FUNCTION_BLOCK SpindleCIA402Velocity IMPLEMENTS SpindleController
VAR
	// CIA402 Control word
	oControlWord AT %Q*: ST_CIA402ControlWord;
	// CIA402 Status word
	iStatusWord AT %I*: UINT;
	// CIA402 actual velocity parameter
	iActualVelocity AT %I* : UDINT;
	// CIA402 target velocity
	oTargetVelocity AT %Q* : INT;
	// Forward/backward is specified by positive or negative speed
	VelocityMultiplier : INT := 1;
END_VAR

(* Return the current speed of the spindle in RPM*)
METHOD GetSpeed : UDINT
GetSpeed := iActualVelocity;
END_METHOD

METHOD GetState : E_CIA402State
VAR CONSTANT
	NotReadyToSwitchOnValue : UINT := 2#0000_0000_0000_0000;
	NotReadyToSwitchOnMask : UINT := 2#0000_0000_0100_1111;
	SwitchOnDisabledValue : UINT := 2#0000_0000_0100_0000;
	SwitchOnDisabledMask : UINT := NotReadyToSwitchOnMask;
	ReadyToSwitchOnValue : UINT := 2#0000_0000_0010_0001;
	ReadyToSwitchOnMask : UINT := 2#0000_0000_0110_1111;
	SwitchedOnValue : UINT := 2#0000_0000_0010_0011;
	SwitchedOnMask : UINT := ReadyToSwitchOnMask;
	OperationEnabledValue : UINT := 2#0000_0000_0010_0111;
	OperationEnabledMask : UINT := ReadyToSwitchOnMask;
	QuickStopActiveValue : UINT := 2#0000_0000_0000_0111;
	QuickStopActiveMask : UINT := ReadyToSwitchOnMask;
	FaultReactionActiveValue : UINT := 2#0000_0000_0000_1111;
	FaultReactionActiveMask : UINT := 2#0000_0000_0100_1111;
	FaultValue : UINT := 2#0000_0000_0000_1000;
	FaultMask : UINT := FaultReactionActiveMask;
END_VAR
IF (iStatusWord AND NotReadyToSwitchOnMask) = NotReadyToSwitchOnValue THEN
	GetState := E_CIA402State.NotReadyToSwitchOn;
ELSIF (iStatusWord AND SwitchOnDisabledMask) = SwitchOnDisabledValue THEN
	GetState := E_CIA402State.SwitchOnDisabled;
ELSIF (iStatusWord AND ReadyToSwitchOnMask) = ReadyToSwitchOnValue THEN
	GetState := E_CIA402State.ReadyToSwitchOn;
ELSIF (iStatusWord AND SwitchedOnMask) = SwitchedOnValue THEN
	GetState := E_CIA402State.SwitchedOn;
ELSIF (iStatusWord AND OperationEnabledMask) = OperationEnabledValue THEN
	GetState := E_CIA402State.OperationEnabled;
ELSIF (iStatusWord AND QuickStopActiveMask) = QuickStopActiveValue THEN
	GetState := E_CIA402State.QuickStopActive;
ELSIF (iStatusWord AND FaultReactionActiveMask) = FaultReactionActiveValue THEN
	GetState := E_CIA402State.FaultReactionActive;
ELSIF (iStatusWord AND FaultMask) = FaultValue THEN
	GetState := E_CIA402State.Fault;
ELSE
	GetState := E_CIA402State.Unknown_State;
END_IF
END_METHOD

METHOD GetStatus : ST_CIA402StatusWord
VAR_INPUT
END_VAR
MEMCPY(ADR(GetStatus), ADR(iStatusWord), SIZEOF(iStatusWord));
END_METHOD

METHOD HasFault : BOOL
VAR_INPUT
END_VAR
HasFault := GetState() = E_CIA402State.Fault OR GetState() = E_CIA402State.FaultReactionActive;
END_METHOD

METHOD Run : BOOL
oControlWord.FaultReset := FALSE;
CASE GetState() OF
	E_CIA402State.SwitchOnDisabled:
		oControlWord.EnableVoltage := TRUE;
	E_CIA402State.ReadyToSwitchOn:
		oControlWord.SwitchOn := TRUE;
	E_CIA402State.SwitchedOn:
		oControlWord.EnableOperation := TRUE;
	// We don't need explicit fault handling. 
	// The fault will cause the controller to tell the drive to stop, 
	// and the stop will take care of the fault reset.
END_CASE
END_METHOD

METHOD SetDirection : BOOL
VAR_INPUT
	(* Set the spindle rotation direction*)
	Reverse	: BOOL;
END_VAR
IF Reverse THEN
	VelocityMultiplier := -1;
ELSE
	VelocityMultiplier := 1;
END_IF
END_METHOD

METHOD SetSpeed : BOOL
VAR_INPUT
	Speed	: UINT;
END_VAR
oTargetVelocity := TO_INT(LIMIT(0, Speed, 32767)) * VelocityMultiplier;
END_METHOD

METHOD Stop : BOOL
oControlWord.FaultReset := FALSE;
CASE GetState() OF
	E_CIA402State.ReadyToSwitchOn:
		oControlWord.EnableVoltage := FALSE;
	E_CIA402State.SwitchedOn:
		oControlWord.SwitchOn := FALSE;
	E_CIA402State.OperationEnabled :
		oControlWord.EnableOperation := FALSE;
	E_CIA402State.Fault : 
		oControlWord.FaultReset := TRUE;
		oControlWord.EnableOperation := FALSE;
		oControlWord.SwitchOn := FALSE;
		oControlWord.EnableVoltage := FALSE;
END_CASE
END_METHOD

END_FUNCTION_BLOCK

(* stored: Version 1.1.0.1, ProductVersion 3.1.4022.18
   POU SpindleCIA402Velocity: Id {02da1002-7a44-4285-a82f-82c9814ffe90}, SpecialFunc None
   Method GetSpeed: Id {f14b85d8-5fa7-4ec3-946f-333b61f1fd83}
   Method GetState: Id {44dd01bf-ad1a-4ea7-92f3-3cd85851766f}
   Method GetStatus: Id {775a00c1-3448-42d6-a5d4-d881a1dfc52a}
   Method HasFault: Id {4a2414af-0535-4476-999a-bd131bda2e15}
   Method Run: Id {ab0e9766-94b8-40b4-9cd9-43564953bb58}
   Method SetDirection: Id {1e6d5a6f-1a48-4509-80a2-a0cebaa7cf13}
   Method SetSpeed: Id {e83d68c2-492a-4627-9d7b-c922fc6b440f}
   Method Stop: Id {9ff9307c-602f-4dec-9675-6a17c3115b1e} *)
